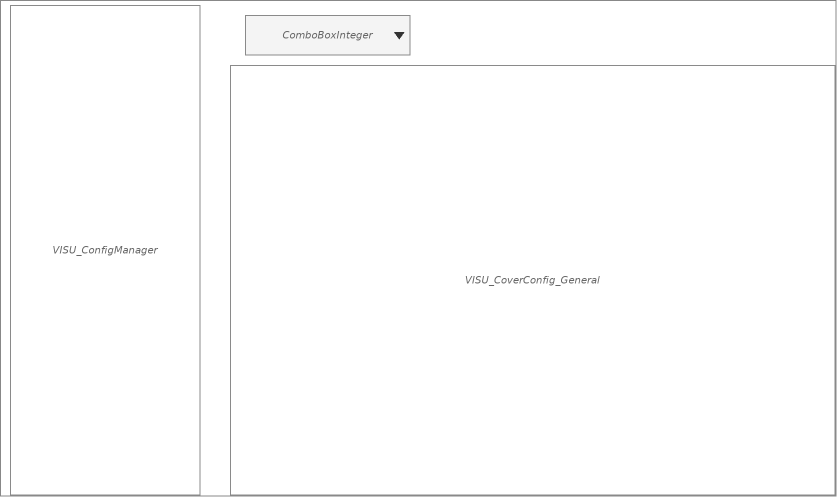
VISUALIZATION VISU_CoverConfig  // 837x497
VAR_IN_OUT
    editableConfig : CoverConfig;
	activeConfig : CoverConfig;
    mgr : ConfigManager;
    mgrWidget : ConfigManagerWidget;
    activeTab : CoverConfigTabs;
END_VAR
    Frame (10,5 190x490)
        shows VISU_ConfigManager(mgr := mgr, widget := mgrWidget)
    ComboBoxInteger (245,15 165x40), variable: activeTab, text list: 'CoverConfigTabsTextList'
    Frame (230,65 605x430), frame switch variable: activeTab
        shows VISU_CoverConfig_General(activeConfig := activeConfig, editableConfig := editableConfig)
        shows VISU_CoverConfig_PanelSet(activeConfig := activeConfig.top, editableConfig := editableConfig.top)
        shows VISU_CoverConfig_PanelSet(activeConfig := activeConfig.bottom, editableConfig := editableConfig.bottom)
        shows VISU_CoverConfig_Panel(activeConfig := activeConfig.top.p1, editableConfig := editableConfig.top.p1)
        shows VISU_CoverConfig_Panel(activeConfig := activeConfig.top.p2, editableConfig := editableConfig.top.p2)
        shows VISU_CoverConfig_Panel(activeConfig := activeConfig.top.p3, editableConfig := editableConfig.top.p3)
        shows VISU_CoverConfig_Panel(activeConfig := activeConfig.top.p4, editableConfig := editableConfig.top.p4)
        shows VISU_CoverConfig_Panel(activeConfig := activeConfig.bottom.p1, editableConfig := editableConfig.bottom.p1)
        shows VISU_CoverConfig_Panel(activeConfig := activeConfig.bottom.p2, editableConfig := editableConfig.bottom.p2)
        shows VISU_CoverConfig_Panel(activeConfig := activeConfig.bottom.p3, editableConfig := editableConfig.bottom.p3)
        shows VISU_CoverConfig_Panel(activeConfig := activeConfig.bottom.p4, editableConfig := editableConfig.bottom.p4)
END_VISUALIZATION

(* stored: Version 1.1.0.1, ProductVersion 3.1.4019.2
   Visu VISU_CoverConfig: Id {f89cb7e3-2baa-4bde-b9b1-0b7042cf4b69} *)
